INTERFACE I_Mc2Settings EXTENDS I_Base

PROPERTY BufferMode : REFERENCE TO tc2_mc2.MC_BufferMode
GET
END_GET
END_PROPERTY

PROPERTY Direction : REFERENCE TO TC2_Mc2.MC_Direction
GET
END_GET
END_PROPERTY

PROPERTY JogMode : REFERENCE TO tc2_mc2.MC_Direction
GET
END_GET
END_PROPERTY

PROPERTY MoveOptions : REFERENCE TO tc2_mc2.ST_MoveOptions
GET
END_GET
END_PROPERTY

END_INTERFACE

(* stored: Version 1.1.0.1, ProductVersion 3.1.4026.20
   Itf I_Mc2Settings: Id {1929287d-762f-4697-b228-a921f106d254}
   Property BufferMode: Id {f9cd230e-b9ee-42f9-bcfc-74725d90540c}
   Get Get: Id {0473fb52-094a-4a04-b49b-da4c5c0db185}
   Property Direction: Id {9ea3bdf2-5d44-4259-96af-5dcfc17c45b6}
   Get Get: Id {b4c90067-f1fa-4d39-9c43-b09bfd3c55fb}
   Property JogMode: Id {1d06df54-3743-4ac5-b830-6ce3d3a8ba36}
   Get Get: Id {0b2fa1ec-77dc-4620-9773-c16cd937bf2c}
   Property MoveOptions: Id {67a6f129-1458-4c62-8a45-ca1066833f2b}
   Get Get: Id {4322c0bb-7fc2-441c-a425-34d56ed57c27} *)
